{attribute 'GeneratedUsingTerminal: EPP1518-0002-0016'}
{attribute addProperty BoxType "EPP1518-0002-0016"}
{attribute addProperty Id "ControlAT %Q*Control_0B2F8B702Set_counter_valueAT %Q*UDINT4"}
{attribute addProperty CRC "1426831071"}
{attribute addProperty Size "6"}
TYPE CNT_Output_Channel_550BB6DF :
STRUCT
	{attribute addProperty Name "Control"}
	Control AT %Q* : Control_0B2F8B70;
	{attribute addProperty Name "Set_counter_value"}
	Set_counter_value AT %Q* : UDINT;
END_STRUCT
END_TYPE

(* stored: Version 1.2.0.0, ProductVersion 3.1.4024.9
   DUT CNT_Output_Channel_550BB6DF: Id {22621a61-33be-4681-874c-824b46c6de69} *)
